FUNCTION_BLOCK FB_KPI_ClearInspectionStatistic
VAR_INPUT
	bExecute						: BOOL;
	stCTDateTime					: ST_SYSTEM_DateTime;	(* CaseTrace date/time structure *)
	nLowerCameraGroupIndex		: INT;
	nUpperCameraGroupIndex		: INT;
END_VAR
VAR_IN_OUT
	stEfficiencyToBeCleared			: ST_KPI_InspectionEfficency;
	stMetsCameras					: ST_NOVRAM_METS_Cameras;
END_VAR
VAR_OUTPUT
	bDone				: BOOL;
END_VAR
VAR
	fbExecute 			: R_TRIG;
	bTimerFlag			: BOOL;
	tofDoneTimer			: TOF;
	nIndex				: INT;

	nCounter				: INT;
END_VAR

(* rising edge of bExecute *)
fbExecute(CLK:= bExecute);

bTimerFlag:=FALSE;

IF fbExecute.Q THEN

	nCounter := nCounter +1;



	MEMSET(ADR(stEfficiencyToBeCleared), 16#00, SIZEOF(stEfficiencyToBeCleared));

	(*stEfficiencyToBeCleared.StartDateTime 			:= F_SYSTEM_SystemTimeAsISO8601(stCTDateTime.sSystemTime, stCTDateTime.sUTCTimeZoneOffset );*)

	IF nLowerCameraGroupIndex > 0 	AND
		nLowerCameraGroupIndex <= nUpperCameraGroupIndex THEN

		FOR nIndex :=nLowerCameraGroupIndex  TO MIN(nUpperCameraGroupIndex, cMAX_CAMERA_NUMBER)  DO
			MEMSET(ADR(stMetsCameras.aCameraEvaluation[nIndex]), 16#00, SIZEOF(stMetsCameras.aCameraEvaluation[nIndex]));
		END_FOR
	END_IF

	bTimerFlag:=TRUE;
END_IF

tofDoneTimer(IN:=bTimerFlag,PT:=t#5s, Q=>bDone);

END_FUNCTION_BLOCK

(* stored: Version 1.1.0.1, ProductVersion 3.1.4024.15
   POU FB_KPI_ClearInspectionStatistic: Id {8b4edb6a-866d-42fc-aba7-ffbd98b3b28b}, SpecialFunc None *)
